Staubli VAL3: refreshPoints.pgx

program refreshPoints(string x_sTrajName)
  local num i
  local num l_nSize
  local string l_sEvent
  local TrajectoryItem l_tTraj
begin
  // load the traj
  call use:listcreate(x_sTrajName)
  //
  call trajType:getSizeItem(false,l_nSize)
  for i=0 to l_nSize-1
    call trajType:getTrajItem(l_tTraj,i)
    l_sEvent=toString("2",i+1)+" "+l_tTraj.comment
    call use:listadd(l_sEvent)
  endFor
  //
end
